FUNCTION_BLOCK UdpSendReceive_Test EXTENDS FB_TestSuite
VAR
	startUdpTest		: BOOL;
	udpTestDone			: BOOL;
	waitListenTestDone	: BOOL;
	tcpServerTestTimeout	: TON := (PT:= T#2M);
	
	udpClient		: TcUdpSendReceive;
	clientAddr		: STRING(15) := '192.168.1.119';
	listenPort		: UINT := 9902;
	sendPort		: UINT := 9901;
	txData			: STRING(25) := 'Hello from PLC UDP client';
	txCounter		: UDINT;
	rxData			: STRING;
	rxCounter		: UDINT;
	methodTimeout	: TON;
END_VAR

udpClient.Run();

IF startUdpTest THEN
	ListenOnUdpPort();
	ReceiveUdpMessage();
	SendUdpMessage();
END_IF

TEST('RunUdpClientTest');
tcpServerTestTimeout(IN:= startUdpTest);
IF udpTestDone THEN
	tcpServerTestTimeout(IN:= FALSE);
	TEST_FINISHED();
ELSIF tcpServerTestTimeout.Q THEN
	AssertFalse(Condition:= tcpServerTestTimeout.Q, Message:= 'UdpClient_Test timed out while running');
	tcpServerTestTimeout(IN:= FALSE);
	TEST_FINISHED();
ELSIF udpClient.Error THEN
	AssertFalse(Condition:= udpClient.Error, Message:= udpClient.GetError);
	tcpServerTestTimeout(IN:= FALSE);
	TEST_FINISHED();
END_IF

METHOD ListenOnUdpPort
VAR_INST
	delay: TIME := T#15S;
END_VAR
IF TEST_ORDERED('ListenOnUdpPort') THEN
	methodTimeout(IN:= TRUE, PT:= delay);
	IF udpClient.StartListen(Port:= listenPort) THEN
		ADSLOGDINT(msgCtrlMask:= ADSLOG_MSGTYPE_LOG, msgFmtStr:= 'UDP client listening on port %d', dintArg:= listenPort);
		waitListenTestDone := TRUE;
		methodTimeout(IN:= FALSE);
		TEST_FINISHED();
	ELSIF methodTimeout.Q THEN
		AssertTrue(Condition:= FALSE, Message:= 'UDP client timed out listening on port');
		methodTimeout(IN:= FALSE);
		TEST_FINISHED();
	END_IF
END_IF
END_METHOD

METHOD ReceiveUdpMessage
VAR_INST
	delay: TIME := T#15S;
END_VAR
IF TEST_ORDERED('ReceiveUdpMessage') THEN
	methodTimeout(IN:= TRUE, PT:= delay);
	IF udpClient.IsDataAvailable THEN
		IF udpClient.Receive(DataPointer:= ADR(rxData), DataLength:= SIZEOF(rxData), ReceivedLength=> rxCounter) THEN
			ADSLOGSTR(msgCtrlMask:= ADSLOG_MSGTYPE_LOG, msgFmtStr:= 'UDP message received: %s', strArg:= rxData);
			AssertTrue(Condition:= rxCounter > 0, Message:= 'The data from the UDP server had a length of zero');
			methodTimeout(IN:= FALSE);
			TEST_FINISHED();
		END_IF
	ELSIF methodTimeout.Q THEN
		AssertTrue(Condition:= FALSE, Message:= 'UDP client timed out waiting for data from the UDP server');
		methodTimeout(IN:= FALSE);
		TEST_FINISHED();
	END_IF
END_IF
END_METHOD

METHOD SendUdpMessage
VAR_INST
	delay: TIME := T#15S;
	i: INT;
END_VAR
IF TEST_ORDERED('SendUdpMessage') THEN
	methodTimeout(IN:= TRUE, PT:= delay);
	IF udpClient.Send(IpAddress:= clientAddr, Port:= sendPort, DataPointer:= ADR(txData), DataLength:= SIZEOF(txData)) THEN
		ADSLOGSTR(msgCtrlMask:= ADSLOG_MSGTYPE_LOG, msgFmtStr:= 'UDP message sent: %s', strArg:= txData);
		udpTestDone := TRUE;
		methodTimeout(IN:= FALSE);
		TEST_FINISHED();
	ELSIF methodTimeout.Q THEN
		AssertTrue(Condition:= FALSE, Message:= 'UDP client timed out sending data to the UDP server');
		methodTimeout(IN:= FALSE);
		TEST_FINISHED();
	END_IF
END_IF
END_METHOD

END_FUNCTION_BLOCK

(* stored: Version 1.1.0.1
   POU UdpSendReceive_Test: Id {c850c202-53d0-0eeb-17a4-d7a260690fc0}, SpecialFunc None
   Method ListenOnUdpPort: Id {a850c202-53d0-0eeb-17a4-d7a260690fc1}
   Method ReceiveUdpMessage: Id {c850c202-53d0-0eeb-17a4-d7a260690fc3}
   Method SendUdpMessage: Id {b850c202-53d0-0eeb-17a4-d7a260690fc2} *)
